(* CODESYS project Liquid_level.project

Project tree, tasks and I/O mapping:
  Device : CODESYS Control Win V3, 3S - Smart Software Solutions GmbH, order no. 305021, version 3.5.7.0
    application Application
      libraries: Standard, * (System)
      task MainTask (cyclic, interval t#20ms, priority 1) calls PLC_PRG
      task VISU_TASK (cyclic, interval 100 ms, priority 31) calls VisuElems.Visu_Prg
      program PLC_PRG [LD]
      visualisation Visualization
  text list GlobalTextList
*)

// Device/Application/PLC_PRG
PROGRAM PLC_PRG
VAR
	man_auto: BOOL;
	low_level: BOOL;
	off_on: BOOL;
	motor: BOOL;
	latch: BOOL;
	high_level: BOOL;
	green: BOOL;
	red: BOOL;
	yellow: BOOL;
END_VAR

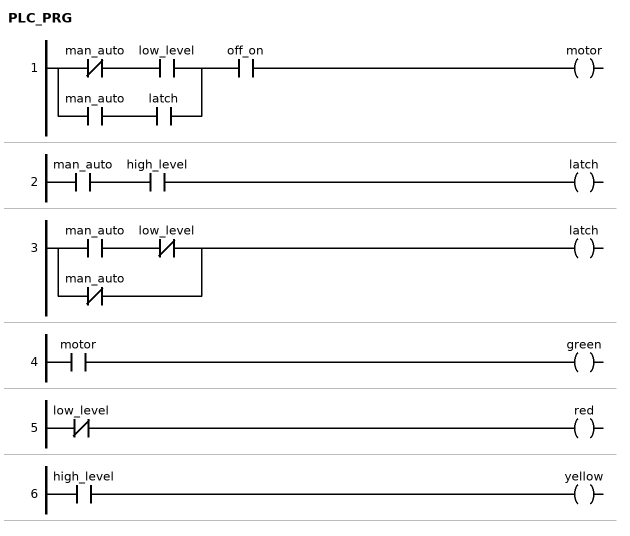
// NETWORK 1
motor := (NOT man_auto AND low_level OR man_auto AND latch) AND off_on;

// NETWORK 2
latch := man_auto AND high_level;

// NETWORK 3
latch := man_auto AND NOT low_level OR NOT man_auto;

// NETWORK 4
green := motor;

// NETWORK 5
red := NOT low_level;

// NETWORK 6
yellow := high_level;

END_PROGRAM

// Device/Application/Visualization
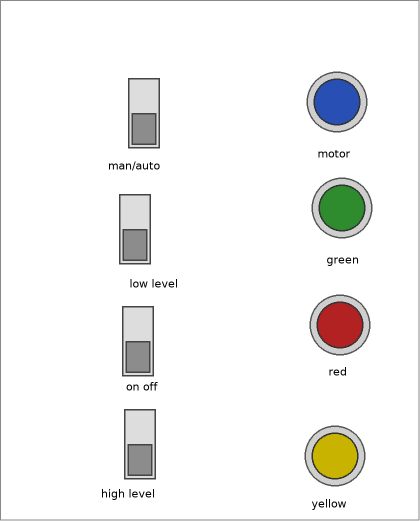
VISUALIZATION Visualization  // 420x521
    Lamp1 (302,67 70x70), variable: PLC_PRG.motor, style: Lamp-Lamp1-Blue
    Lamp1 (307,173 70x70), variable: PLC_PRG.green, style: Lamp-Lamp1-Green
    Lamp1 (305,290 70x70), variable: PLC_PRG.red, style: Lamp-Lamp1-Red
    Lamp1 (300,421 70x70), variable: PLC_PRG.yellow, style: Lamp-Lamp1-Yellow
    DipSwitch (109,78 70x70), variable: PLC_PRG.man_auto, behaviour: TOGGLE, style: Switch-DipSwitch-Gray
    DipSwitch (100,194 70x70), variable: PLC_PRG.low_level, behaviour: TOGGLE, style: Switch-DipSwitch-Gray
    DipSwitch (103,306 70x70), variable: PLC_PRG.off_on, behaviour: TOGGLE, style: Switch-DipSwitch-Gray
    DipSwitch (105,409 70x70), variable: PLC_PRG.high_level, behaviour: TOGGLE, style: Switch-DipSwitch-Gray
    Label (59,151 150x30), "man/auto"
    Label (79,269 150x30), "low level"
    Label (67,372 150x30), "on off"
    Label (53,479 150x30), "high level"
    Label (259,139 150x30), "motor"
    Label (268,245 150x30), "green"
    Label (263,357 150x30), "red"
    Label (254,489 150x30), "yellow"
END_VISUALIZATION
